{attribute 'GeneratedUsingTerminal: CX5130 EtherCAT slave-1b82-0016'}
{attribute addProperty BoxType "CX5130 EtherCAT slave-1b82-0016"}
{attribute addProperty Id "EtcSlaveTerminalBaseIO_InputsEMPTY_STRUCTURE0Device_Status_MappingAT %I*Device_Status_Mapping_61F790772IO_OutputsEMPTY_STRUCTURE0WcStateAT %I*WcState_9091E0EB2InfoDataAT %I*InfoData_90184F0C16"}
{attribute addProperty CRC "143137934"}
{attribute addProperty Size "20"}
TYPE CX5130_EtherCAT_slave_08881C8E EXTENDS EtcSlaveTerminalBase :
STRUCT
	{attribute addProperty Name "IO_Inputs"}
	IO_Inputs : EMPTY_STRUCTURE;
	{attribute addProperty Name "Device_Status_Mapping"}
	Device_Status_Mapping : Device_Status_Mapping_61F79077;
	{attribute addProperty Name "IO_Outputs"}
	IO_Outputs : EMPTY_STRUCTURE;
	{attribute addProperty Name "WcState"}
	WcState : WcState_9091E0EB;
	{attribute addProperty Name "InfoData"}
	InfoData : InfoData_90184F0C;
END_STRUCT
END_TYPE

(* stored: Version 1.2.0.0, ProductVersion 3.1.4024.9
   DUT CX5130_EtherCAT_slave_08881C8E: Id {096cdaaf-bf2c-4980-a257-d05e87635dce} *)
